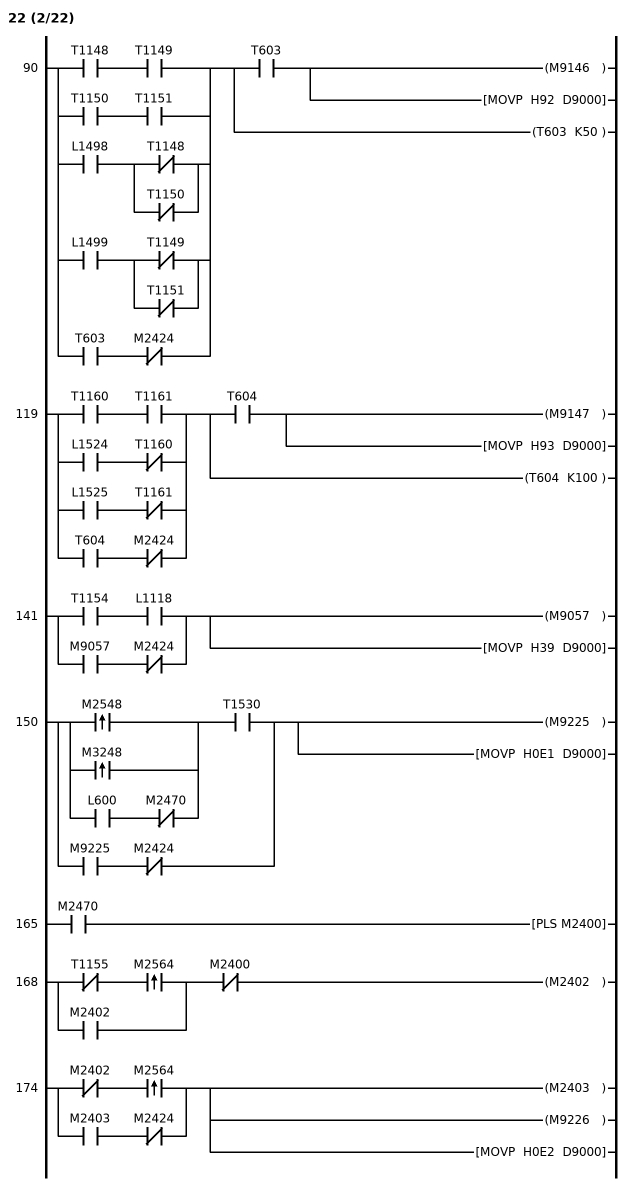
90    LD      T1148
      AND     T1149
      LD      T1150
      AND     T1151
      ORB
      LD      L1498
      LDI     T1148
      ORI     T1150
      ANB
      ORB
      LD      L1499
      LDI     T1149
      ORI     T1151
      ANB
      ORB
      LD      T603
      ANI     M2424
      ORB
      MPS
      AND     T603
      OUT     M9146
      MOVP    H92 D9000
      MPP
      OUT     T603 K50
119   LD      T1160
      AND     T1161
      LD      L1524
      ANI     T1160
      ORB
      LD      L1525
      ANI     T1161
      ORB
      LD      T604
      ANI     M2424
      ORB
      MPS
      AND     T604
      OUT     M9147
      MOVP    H93 D9000
      MPP
      OUT     T604 K100
141   LD      T1154
      AND     L1118
      LD      M9057
      ANI     M2424
      ORB
      OUT     M9057
      MOVP    H39 D9000
150   LDP     M2548
      ORP     M3248
      LD      L600
      ANI     M2470
      ORB
      AND     T1530
      LD      M9225
      ANI     M2424
      ORB
      OUT     M9225
      MOVP    H0E1 D9000
165   LD      M2470
      PLS     M2400
168   LDI     T1155
      ANDP    M2564
      OR      M2402
      ANI     M2400
      OUT     M2402
174   LDI     M2402
      ANDP    M2564
      LD      M2403
      ANI     M2424
      ORB
      OUT     M2403
      OUT     M9226
      MOVP    H0E2 D9000
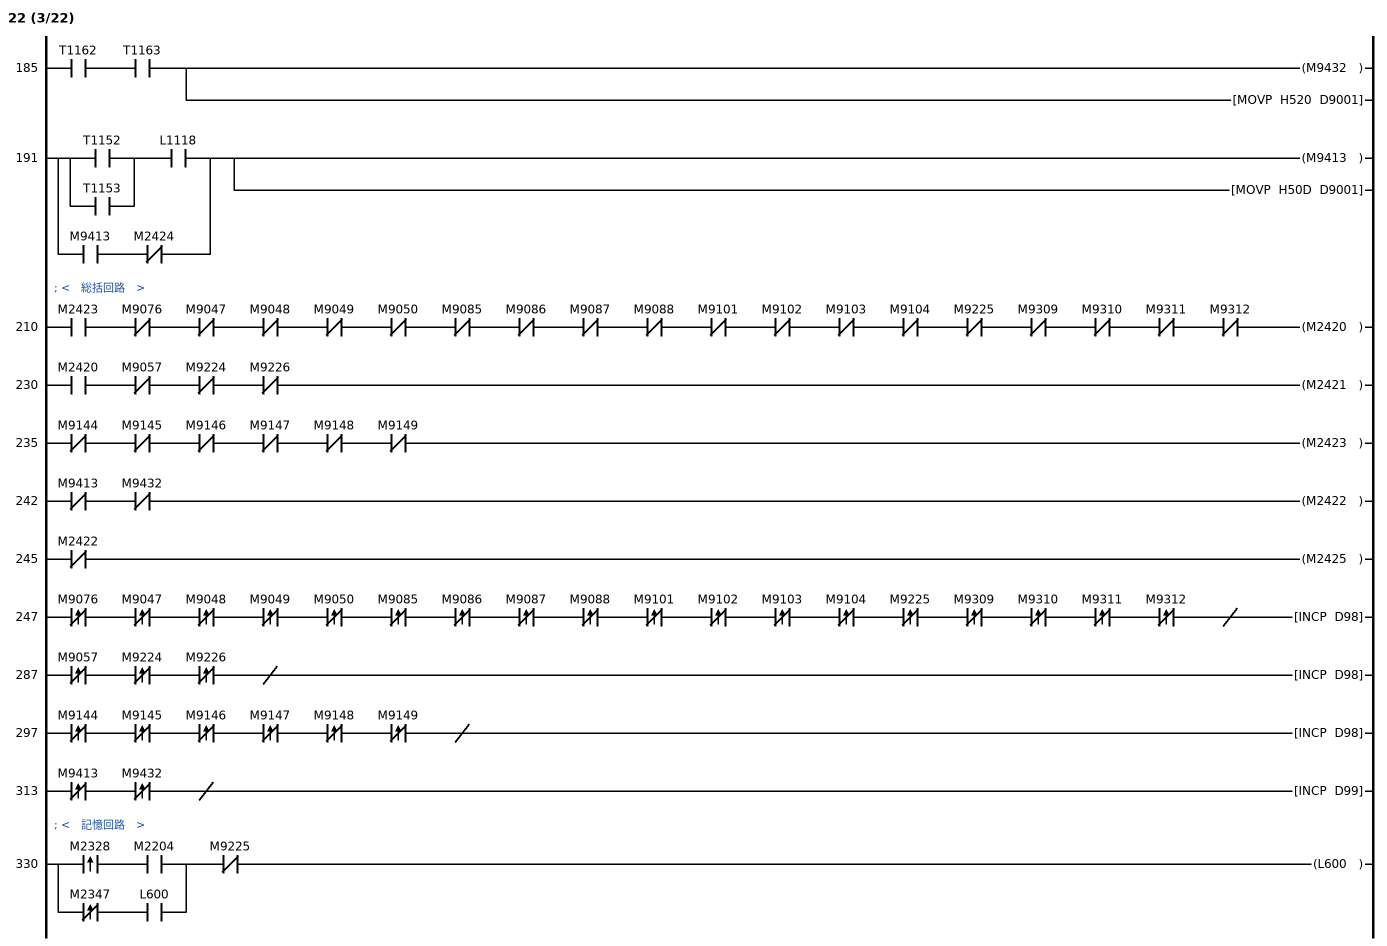
185   LD      T1162
      AND     T1163
      OUT     M9432
      MOVP    H520 D9001
191   LD      T1152
      OR      T1153
      AND     L1118
      LD      M9413
      ANI     M2424
      ORB
      OUT     M9413
      MOVP    H50D D9001
; <　総括回路　>
210   LD      M2423
      ANI     M9076
      ANI     M9047
      ANI     M9048
      ANI     M9049
      ANI     M9050
      ANI     M9085
      ANI     M9086
      ANI     M9087
      ANI     M9088
      ANI     M9101
      ANI     M9102
      ANI     M9103
      ANI     M9104
      ANI     M9225
      ANI     M9309
      ANI     M9310
      ANI     M9311
      ANI     M9312
      OUT     M2420
230   LD      M2420
      ANI     M9057
      ANI     M9224
      ANI     M9226
      OUT     M2421
235   LDI     M9144
      ANI     M9145
      ANI     M9146
      ANI     M9147
      ANI     M9148
      ANI     M9149
      OUT     M2423
242   LDI     M9413
      ANI     M9432
      OUT     M2422
245   LDI     M2422
      OUT     M2425
247   LDPI    M9076
      ANDPI   M9047
      ANDPI   M9048
      ANDPI   M9049
      ANDPI   M9050
      ANDPI   M9085
      ANDPI   M9086
      ANDPI   M9087
      ANDPI   M9088
      ANDPI   M9101
      ANDPI   M9102
      ANDPI   M9103
      ANDPI   M9104
      ANDPI   M9225
      ANDPI   M9309
      ANDPI   M9310
      ANDPI   M9311
      ANDPI   M9312
      INV
      INCP    D98
287   LDPI    M9057
      ANDPI   M9224
      ANDPI   M9226
      INV
      INCP    D98
297   LDPI    M9144
      ANDPI   M9145
      ANDPI   M9146
      ANDPI   M9147
      ANDPI   M9148
      ANDPI   M9149
      INV
      INCP    D98
313   LDPI    M9413
      ANDPI   M9432
      INV
      INCP    D99
; <　記憶回路　>
330   LDP     M2328
      AND     M2204
      LDPI    M2347
      AND     L600
      ORB
      ANI     M9225
      OUT     L600
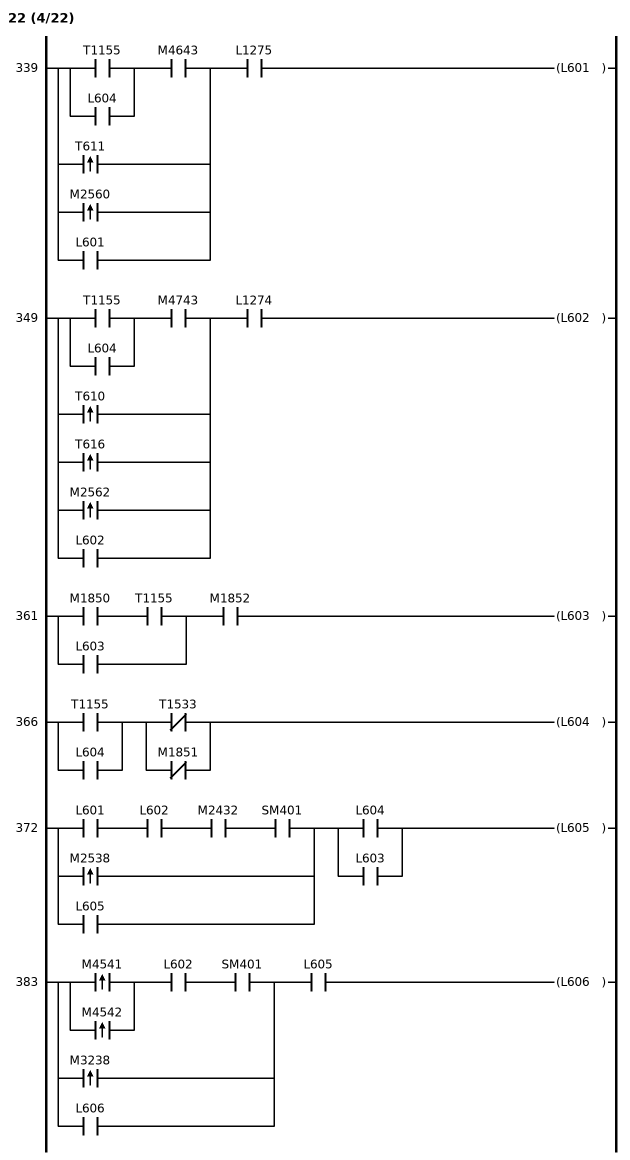
339   LD      T1155
      OR      L604
      AND     M4643
      ORP     T611
      ORP     M2560
      OR      L601
      AND     L1275
      OUT     L601
349   LD      T1155
      OR      L604
      AND     M4743
      ORP     T610
      ORP     T616
      ORP     M2562
      OR      L602
      AND     L1274
      OUT     L602
361   LD      M1850
      AND     T1155
      OR      L603
      AND     M1852
      OUT     L603
366   LD      T1155
      OR      L604
      LDI     T1533
      ORI     M1851
      ANB
      OUT     L604
372   LD      L601
      AND     L602
      AND     M2432
      AND     SM401
      ORP     M2538
      OR      L605
      LD      L604
      OR      L603
      ANB
      OUT     L605
383   LDP     M4541
      ORP     M4542
      AND     L602
      AND     SM401
      ORP     M3238
      OR      L606
      AND     L605
      OUT     L606
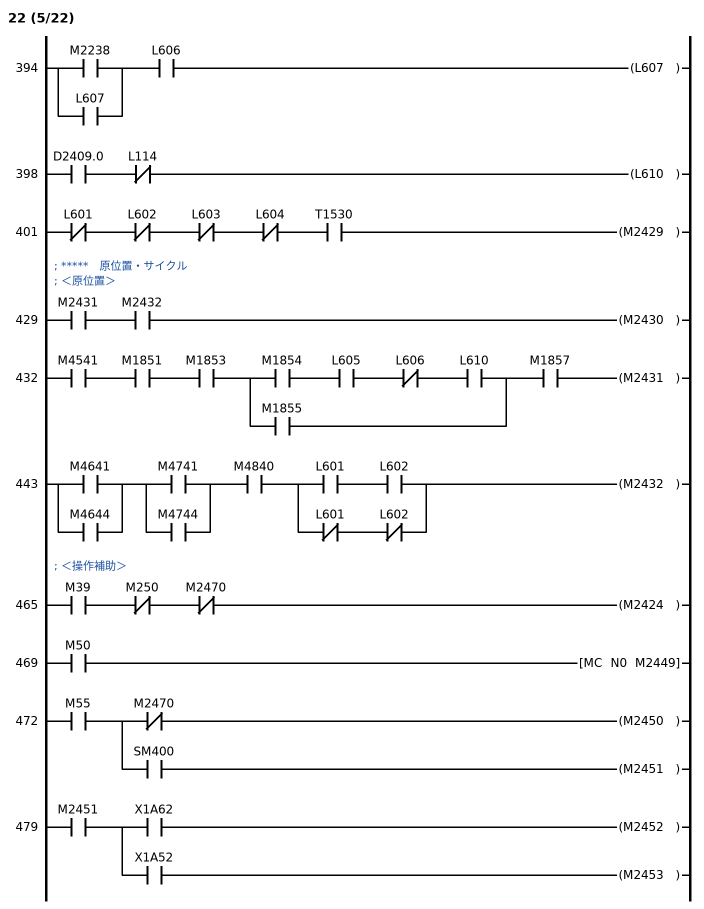
394   LD      M2238
      OR      L607
      AND     L606
      OUT     L607
398   LD      D2409.0
      ANI     L114
      OUT     L610
401   LDI     L601
      ANI     L602
      ANI     L603
      ANI     L604
      AND     T1530
      OUT     M2429
; *****　原位置・サイクル
; ＜原位置＞
429   LD      M2431
      AND     M2432
      OUT     M2430
432   LD      M4541
      AND     M1851
      AND     M1853
      LD      M1854
      AND     L605
      ANI     L606
      AND     L610
      OR      M1855
      ANB
      AND     M1857
      OUT     M2431
443   LD      M4641
      OR      M4644
      LD      M4741
      OR      M4744
      ANB
      AND     M4840
      LD      L601
      AND     L602
      LDI     L601
      ANI     L602
      ORB
      ANB
      OUT     M2432
; ＜操作補助＞
465   LD      M39
      ANI     M250
      ANI     M2470
      OUT     M2424
469   LD      M50
      MC      N0 M2449
472   LD      M55
      MPS
      ANI     M2470
      OUT     M2450
      MPP
      AND     SM400
      OUT     M2451
479   LD      M2451
      MPS
      AND     X1A62
      OUT     M2452
      MPP
      AND     X1A52
      OUT     M2453
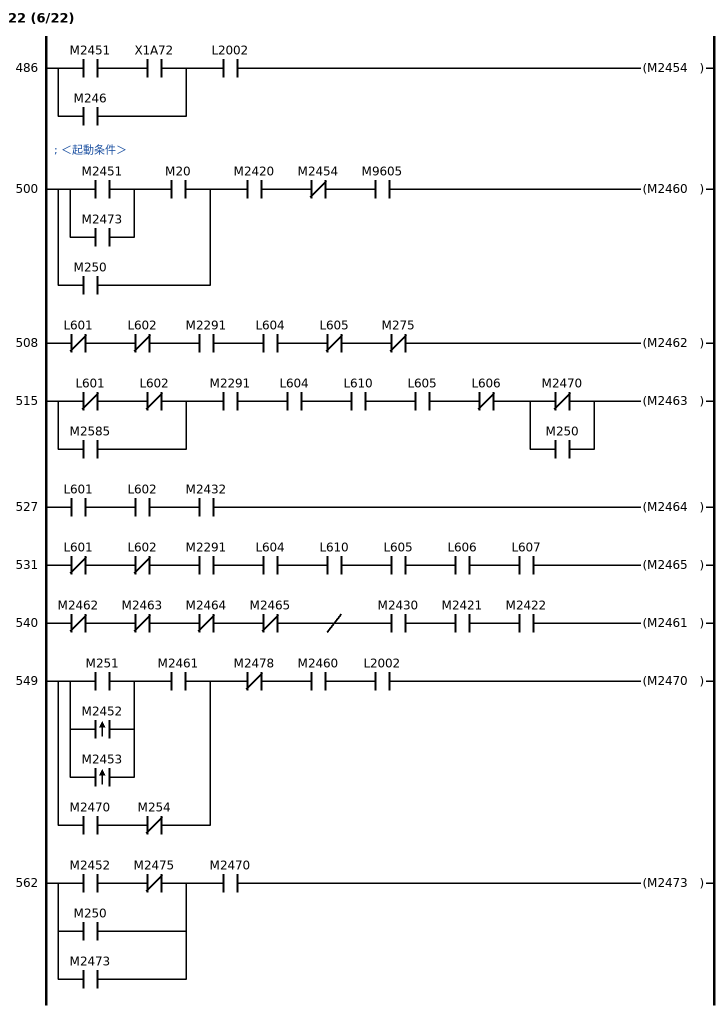
486   LD      M2451
      AND     X1A72
      OR      M246
      AND     L2002
      OUT     M2454
; ＜起動条件＞
500   LD      M2451
      OR      M2473
      AND     M20
      OR      M250
      AND     M2420
      ANI     M2454
      AND     M9605
      OUT     M2460
508   LDI     L601
      ANI     L602
      AND     M2291
      AND     L604
      ANI     L605
      ANI     M275
      OUT     M2462
515   LDI     L601
      ANI     L602
      OR      M2585
      AND     M2291
      AND     L604
      AND     L610
      AND     L605
      ANI     L606
      LDI     M2470
      OR      M250
      ANB
      OUT     M2463
527   LD      L601
      AND     L602
      AND     M2432
      OUT     M2464
531   LDI     L601
      ANI     L602
      AND     M2291
      AND     L604
      AND     L610
      AND     L605
      AND     L606
      AND     L607
      OUT     M2465
540   LDI     M2462
      ANI     M2463
      ANI     M2464
      ANI     M2465
      INV
      AND     M2430
      AND     M2421
      AND     M2422
      OUT     M2461
549   LD      M251
      ORP     M2452
      ORP     M2453
      AND     M2461
      LD      M2470
      ANI     M254
      ORB
      ANI     M2478
      AND     M2460
      AND     L2002
      OUT     M2470
562   LD      M2452
      ANI     M2475
      OR      M250
      OR      M2473
      AND     M2470
      OUT     M2473
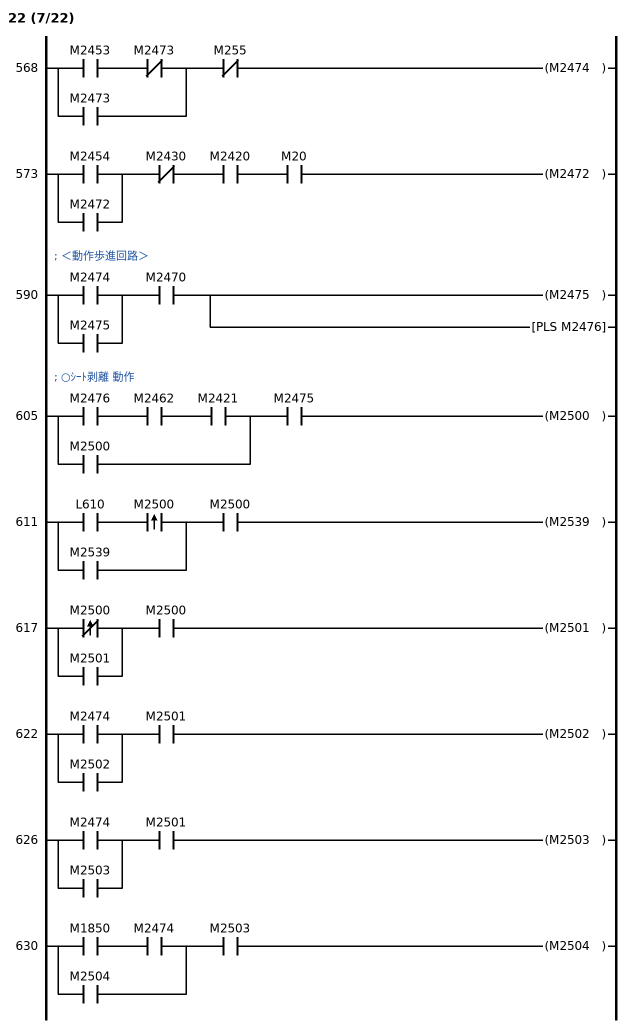
568   LD      M2453
      ANI     M2473
      OR      M2473
      ANI     M255
      OUT     M2474
573   LD      M2454
      OR      M2472
      ANI     M2430
      AND     M2420
      AND     M20
      OUT     M2472
; ＜動作歩進回路＞
590   LD      M2474
      OR      M2475
      AND     M2470
      OUT     M2475
      PLS     M2476
; ○ｼｰﾄ剥離 動作
605   LD      M2476
      AND     M2462
      AND     M2421
      OR      M2500
      AND     M2475
      OUT     M2500
611   LD      L610
      ANDP    M2500
      OR      M2539
      AND     M2500
      OUT     M2539
617   LDPI    M2500
      OR      M2501
      AND     M2500
      OUT     M2501
622   LD      M2474
      OR      M2502
      AND     M2501
      OUT     M2502
626   LD      M2474
      OR      M2503
      AND     M2501
      OUT     M2503
630   LD      M1850
      AND     M2474
      OR      M2504
      AND     M2503
      OUT     M2504
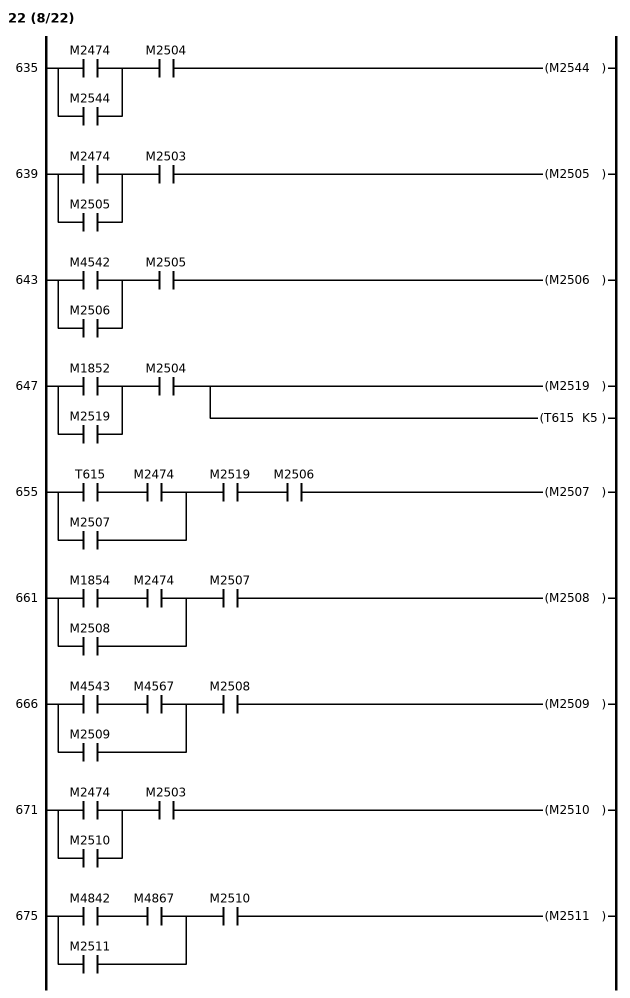
635   LD      M2474
      OR      M2544
      AND     M2504
      OUT     M2544
639   LD      M2474
      OR      M2505
      AND     M2503
      OUT     M2505
643   LD      M4542
      OR      M2506
      AND     M2505
      OUT     M2506
647   LD      M1852
      OR      M2519
      AND     M2504
      OUT     M2519
      OUT     T615 K5
655   LD      T615
      AND     M2474
      OR      M2507
      AND     M2519
      AND     M2506
      OUT     M2507
661   LD      M1854
      AND     M2474
      OR      M2508
      AND     M2507
      OUT     M2508
666   LD      M4543
      AND     M4567
      OR      M2509
      AND     M2508
      OUT     M2509
671   LD      M2474
      OR      M2510
      AND     M2503
      OUT     M2510
675   LD      M4842
      AND     M4867
      OR      M2511
      AND     M2510
      OUT     M2511
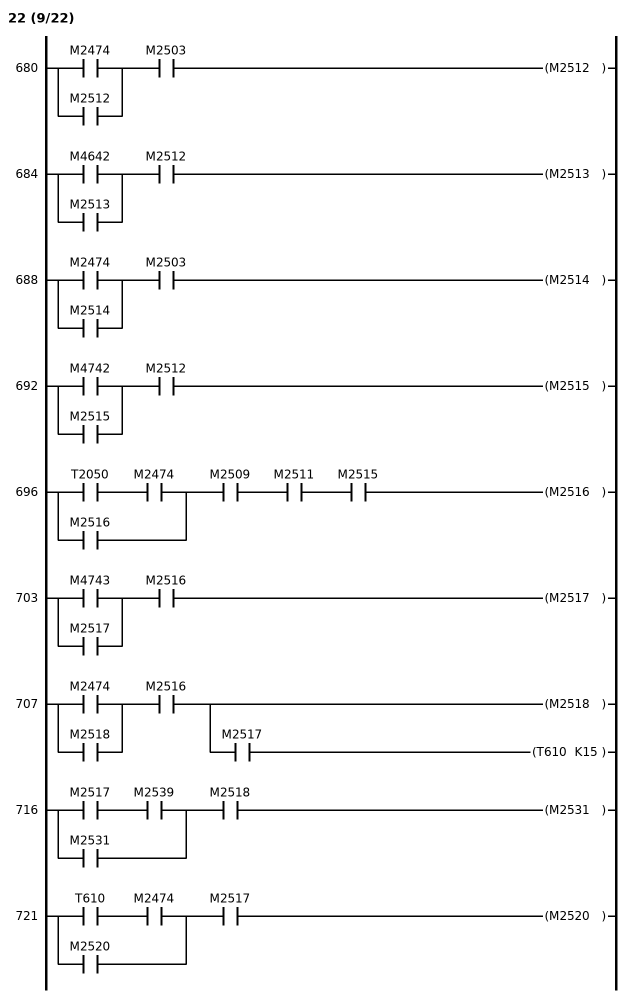
680   LD      M2474
      OR      M2512
      AND     M2503
      OUT     M2512
684   LD      M4642
      OR      M2513
      AND     M2512
      OUT     M2513
688   LD      M2474
      OR      M2514
      AND     M2503
      OUT     M2514
692   LD      M4742
      OR      M2515
      AND     M2512
      OUT     M2515
696   LD      T2050
      AND     M2474
      OR      M2516
      AND     M2509
      AND     M2511
      AND     M2515
      OUT     M2516
703   LD      M4743
      OR      M2517
      AND     M2516
      OUT     M2517
707   LD      M2474
      OR      M2518
      AND     M2516
      OUT     M2518
      AND     M2517
      OUT     T610 K15
716   LD      M2517
      AND     M2539
      OR      M2531
      AND     M2518
      OUT     M2531
721   LD      T610
      AND     M2474
      OR      M2520
      AND     M2517
      OUT     M2520
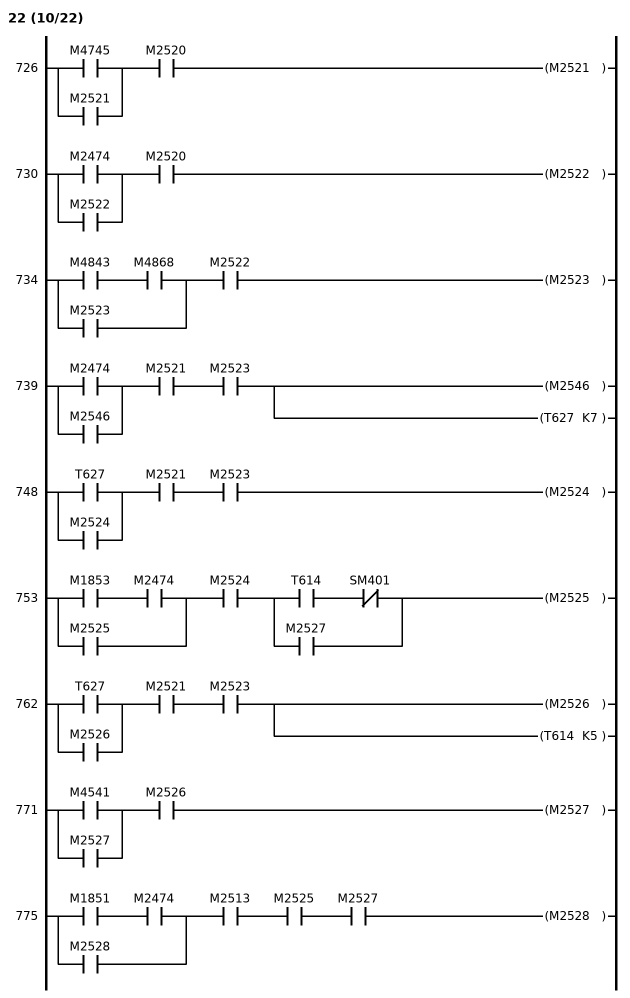
726   LD      M4745
      OR      M2521
      AND     M2520
      OUT     M2521
730   LD      M2474
      OR      M2522
      AND     M2520
      OUT     M2522
734   LD      M4843
      AND     M4868
      OR      M2523
      AND     M2522
      OUT     M2523
739   LD      M2474
      OR      M2546
      AND     M2521
      AND     M2523
      OUT     M2546
      OUT     T627 K7
748   LD      T627
      OR      M2524
      AND     M2521
      AND     M2523
      OUT     M2524
753   LD      M1853
      AND     M2474
      OR      M2525
      AND     M2524
      LD      T614
      ANI     SM401
      OR      M2527
      ANB
      OUT     M2525
762   LD      T627
      OR      M2526
      AND     M2521
      AND     M2523
      OUT     M2526
      OUT     T614 K5
771   LD      M4541
      OR      M2527
      AND     M2526
      OUT     M2527
775   LD      M1851
      AND     M2474
      OR      M2528
      AND     M2513
      AND     M2525
      AND     M2527
      OUT     M2528
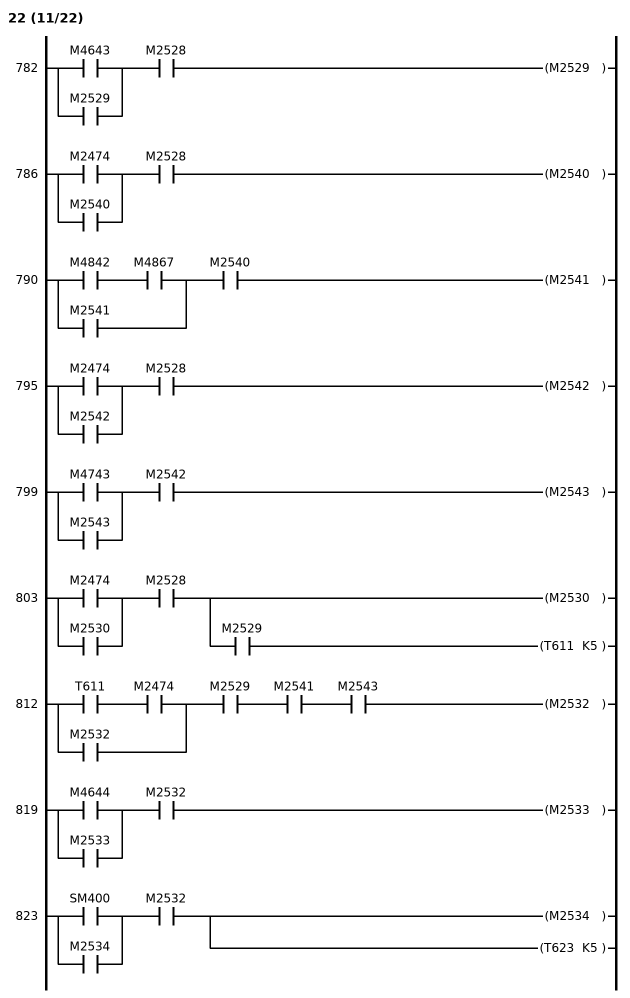
782   LD      M4643
      OR      M2529
      AND     M2528
      OUT     M2529
786   LD      M2474
      OR      M2540
      AND     M2528
      OUT     M2540
790   LD      M4842
      AND     M4867
      OR      M2541
      AND     M2540
      OUT     M2541
795   LD      M2474
      OR      M2542
      AND     M2528
      OUT     M2542
799   LD      M4743
      OR      M2543
      AND     M2542
      OUT     M2543
803   LD      M2474
      OR      M2530
      AND     M2528
      OUT     M2530
      AND     M2529
      OUT     T611 K5
812   LD      T611
      AND     M2474
      OR      M2532
      AND     M2529
      AND     M2541
      AND     M2543
      OUT     M2532
819   LD      M4644
      OR      M2533
      AND     M2532
      OUT     M2533
823   LD      SM400
      OR      M2534
      AND     M2532
      OUT     M2534
      OUT     T623 K5
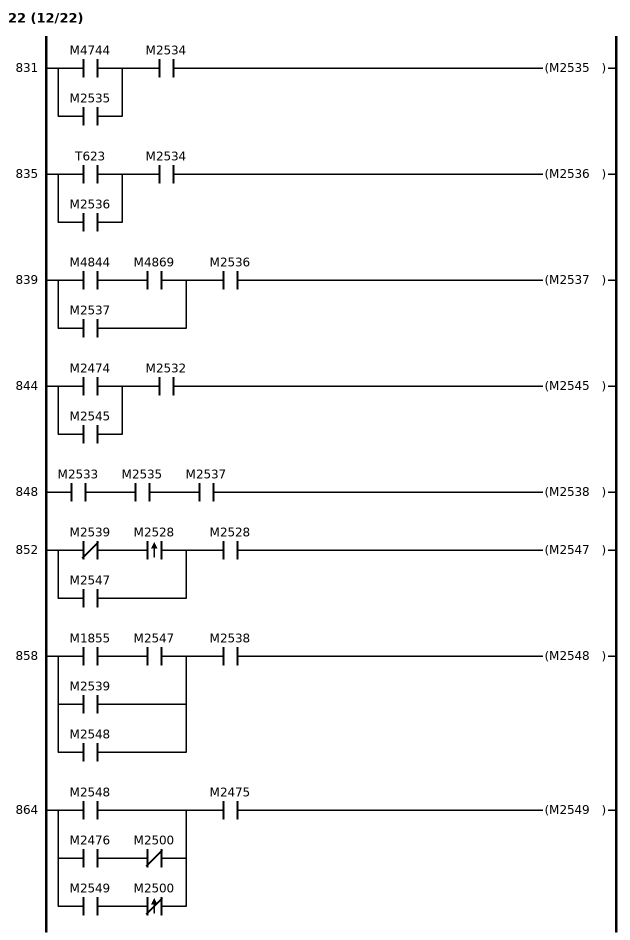
831   LD      M4744
      OR      M2535
      AND     M2534
      OUT     M2535
835   LD      T623
      OR      M2536
      AND     M2534
      OUT     M2536
839   LD      M4844
      AND     M4869
      OR      M2537
      AND     M2536
      OUT     M2537
844   LD      M2474
      OR      M2545
      AND     M2532
      OUT     M2545
848   LD      M2533
      AND     M2535
      AND     M2537
      OUT     M2538
852   LDI     M2539
      ANDP    M2528
      OR      M2547
      AND     M2528
      OUT     M2547
858   LD      M1855
      AND     M2547
      OR      M2539
      OR      M2548
      AND     M2538
      OUT     M2548
864   LD      M2548
      LD      M2476
      ANI     M2500
      ORB
      LD      M2549
      ANDPI   M2500
      ORB
      AND     M2475
      OUT     M2549
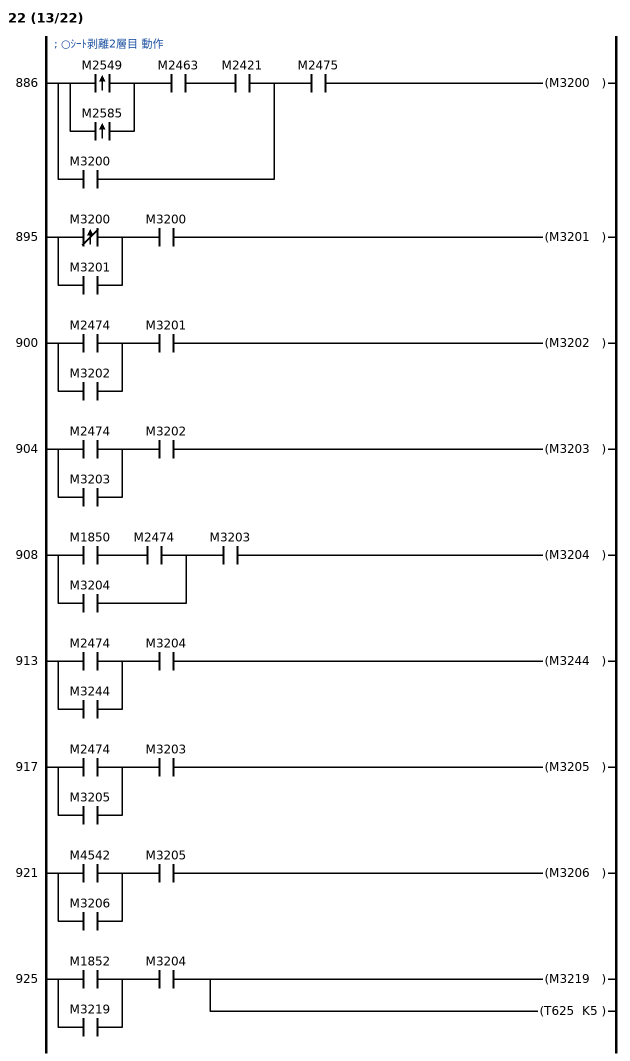
; ○ｼｰﾄ剥離2層目 動作
886   LDP     M2549
      ORP     M2585
      AND     M2463
      AND     M2421
      OR      M3200
      AND     M2475
      OUT     M3200
895   LDPI    M3200
      OR      M3201
      AND     M3200
      OUT     M3201
900   LD      M2474
      OR      M3202
      AND     M3201
      OUT     M3202
904   LD      M2474
      OR      M3203
      AND     M3202
      OUT     M3203
908   LD      M1850
      AND     M2474
      OR      M3204
      AND     M3203
      OUT     M3204
913   LD      M2474
      OR      M3244
      AND     M3204
      OUT     M3244
917   LD      M2474
      OR      M3205
      AND     M3203
      OUT     M3205
921   LD      M4542
      OR      M3206
      AND     M3205
      OUT     M3206
925   LD      M1852
      OR      M3219
      AND     M3204
      OUT     M3219
      OUT     T625 K5
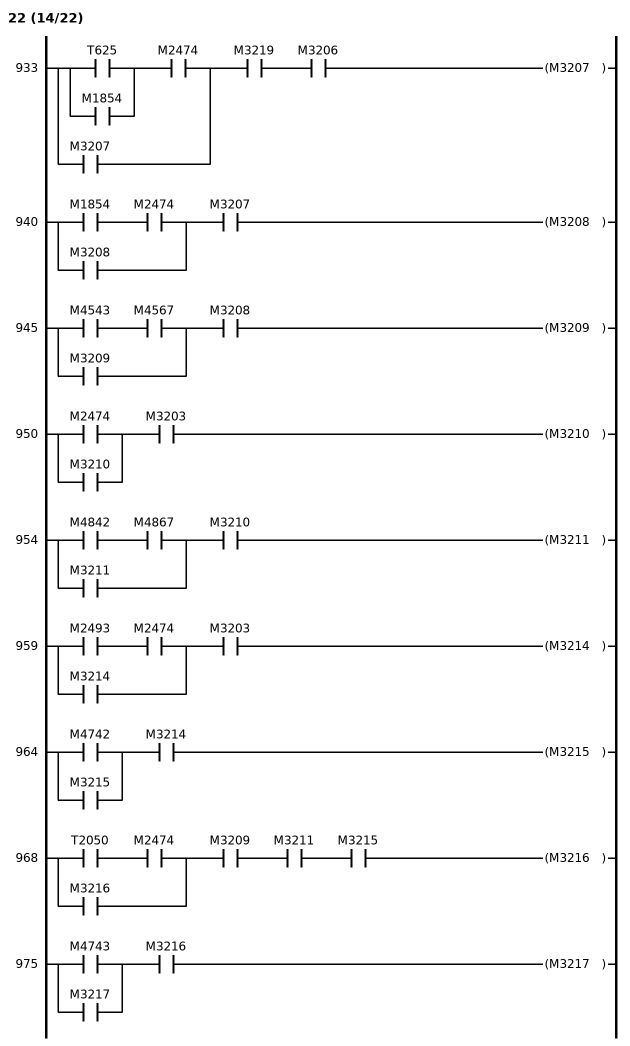
933   LD      T625
      OR      M1854
      AND     M2474
      OR      M3207
      AND     M3219
      AND     M3206
      OUT     M3207
940   LD      M1854
      AND     M2474
      OR      M3208
      AND     M3207
      OUT     M3208
945   LD      M4543
      AND     M4567
      OR      M3209
      AND     M3208
      OUT     M3209
950   LD      M2474
      OR      M3210
      AND     M3203
      OUT     M3210
954   LD      M4842
      AND     M4867
      OR      M3211
      AND     M3210
      OUT     M3211
959   LD      M2493
      AND     M2474
      OR      M3214
      AND     M3203
      OUT     M3214
964   LD      M4742
      OR      M3215
      AND     M3214
      OUT     M3215
968   LD      T2050
      AND     M2474
      OR      M3216
      AND     M3209
      AND     M3211
      AND     M3215
      OUT     M3216
975   LD      M4743
      OR      M3217
      AND     M3216
      OUT     M3217
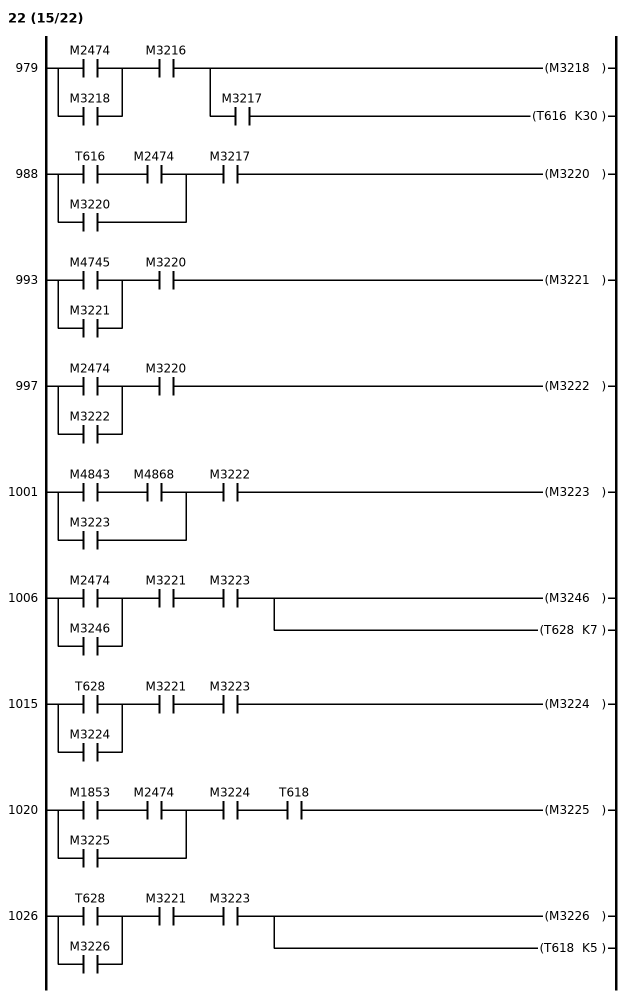
979   LD      M2474
      OR      M3218
      AND     M3216
      OUT     M3218
      AND     M3217
      OUT     T616 K30
988   LD      T616
      AND     M2474
      OR      M3220
      AND     M3217
      OUT     M3220
993   LD      M4745
      OR      M3221
      AND     M3220
      OUT     M3221
997   LD      M2474
      OR      M3222
      AND     M3220
      OUT     M3222
1001  LD      M4843
      AND     M4868
      OR      M3223
      AND     M3222
      OUT     M3223
1006  LD      M2474
      OR      M3246
      AND     M3221
      AND     M3223
      OUT     M3246
      OUT     T628 K7
1015  LD      T628
      OR      M3224
      AND     M3221
      AND     M3223
      OUT     M3224
1020  LD      M1853
      AND     M2474
      OR      M3225
      AND     M3224
      AND     T618
      OUT     M3225
1026  LD      T628
      OR      M3226
      AND     M3221
      AND     M3223
      OUT     M3226
      OUT     T618 K5
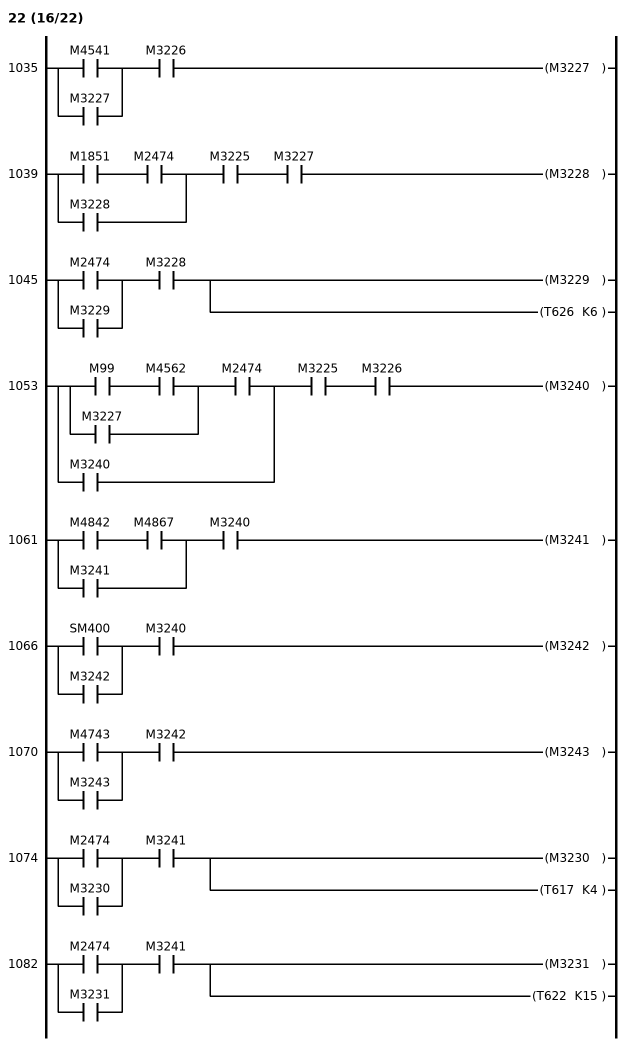
1035  LD      M4541
      OR      M3227
      AND     M3226
      OUT     M3227
1039  LD      M1851
      AND     M2474
      OR      M3228
      AND     M3225
      AND     M3227
      OUT     M3228
1045  LD      M2474
      OR      M3229
      AND     M3228
      OUT     M3229
      OUT     T626 K6
1053  LD      M99
      AND     M4562
      OR      M3227
      AND     M2474
      OR      M3240
      AND     M3225
      AND     M3226
      OUT     M3240
1061  LD      M4842
      AND     M4867
      OR      M3241
      AND     M3240
      OUT     M3241
1066  LD      SM400
      OR      M3242
      AND     M3240
      OUT     M3242
1070  LD      M4743
      OR      M3243
      AND     M3242
      OUT     M3243
1074  LD      M2474
      OR      M3230
      AND     M3241
      OUT     M3230
      OUT     T617 K4
1082  LD      M2474
      OR      M3231
      AND     M3241
      OUT     M3231
      OUT     T622 K15
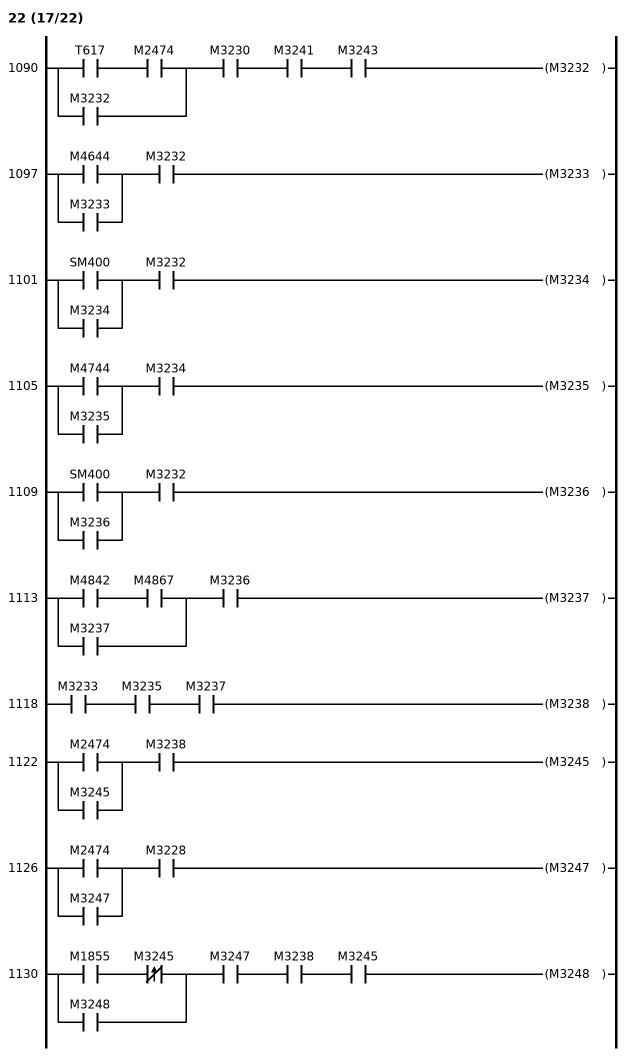
1090  LD      T617
      AND     M2474
      OR      M3232
      AND     M3230
      AND     M3241
      AND     M3243
      OUT     M3232
1097  LD      M4644
      OR      M3233
      AND     M3232
      OUT     M3233
1101  LD      SM400
      OR      M3234
      AND     M3232
      OUT     M3234
1105  LD      M4744
      OR      M3235
      AND     M3234
      OUT     M3235
1109  LD      SM400
      OR      M3236
      AND     M3232
      OUT     M3236
1113  LD      M4842
      AND     M4867
      OR      M3237
      AND     M3236
      OUT     M3237
1118  LD      M3233
      AND     M3235
      AND     M3237
      OUT     M3238
1122  LD      M2474
      OR      M3245
      AND     M3238
      OUT     M3245
1126  LD      M2474
      OR      M3247
      AND     M3228
      OUT     M3247
1130  LD      M1855
      ANDPI   M3245
      OR      M3248
      AND     M3247
      AND     M3238
      AND     M3245
      OUT     M3248
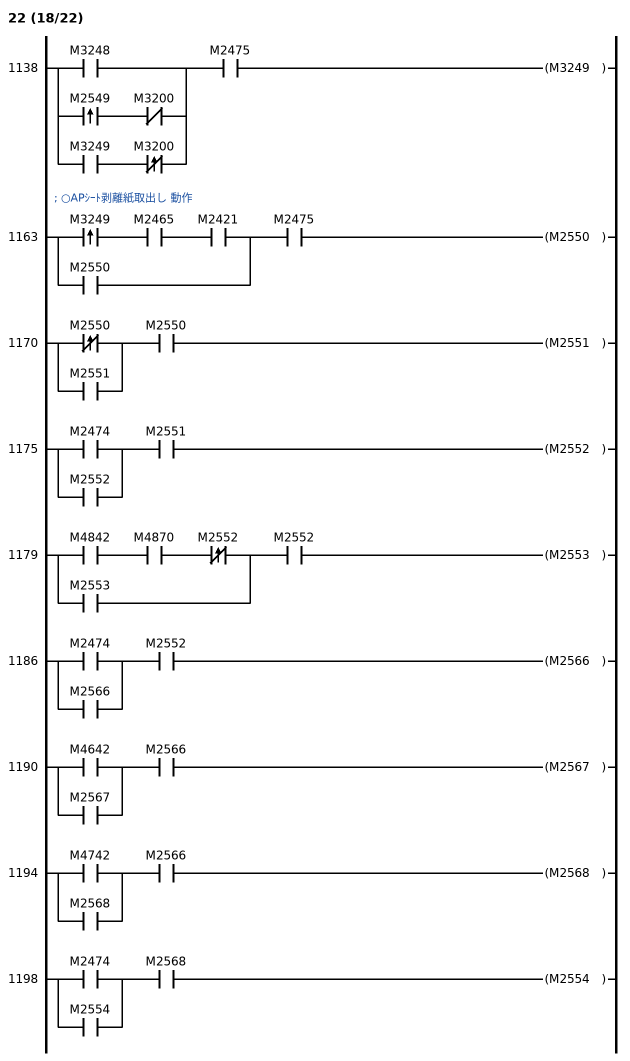
1138  LD      M3248
      LDP     M2549
      ANI     M3200
      ORB
      LD      M3249
      ANDPI   M3200
      ORB
      AND     M2475
      OUT     M3249
; ○APｼｰﾄ剥離紙取出し 動作
1163  LDP     M3249
      AND     M2465
      AND     M2421
      OR      M2550
      AND     M2475
      OUT     M2550
1170  LDPI    M2550
      OR      M2551
      AND     M2550
      OUT     M2551
1175  LD      M2474
      OR      M2552
      AND     M2551
      OUT     M2552
1179  LD      M4842
      AND     M4870
      ANDPI   M2552
      OR      M2553
      AND     M2552
      OUT     M2553
1186  LD      M2474
      OR      M2566
      AND     M2552
      OUT     M2566
1190  LD      M4642
      OR      M2567
      AND     M2566
      OUT     M2567
1194  LD      M4742
      OR      M2568
      AND     M2566
      OUT     M2568
1198  LD      M2474
      OR      M2554
      AND     M2568
      OUT     M2554
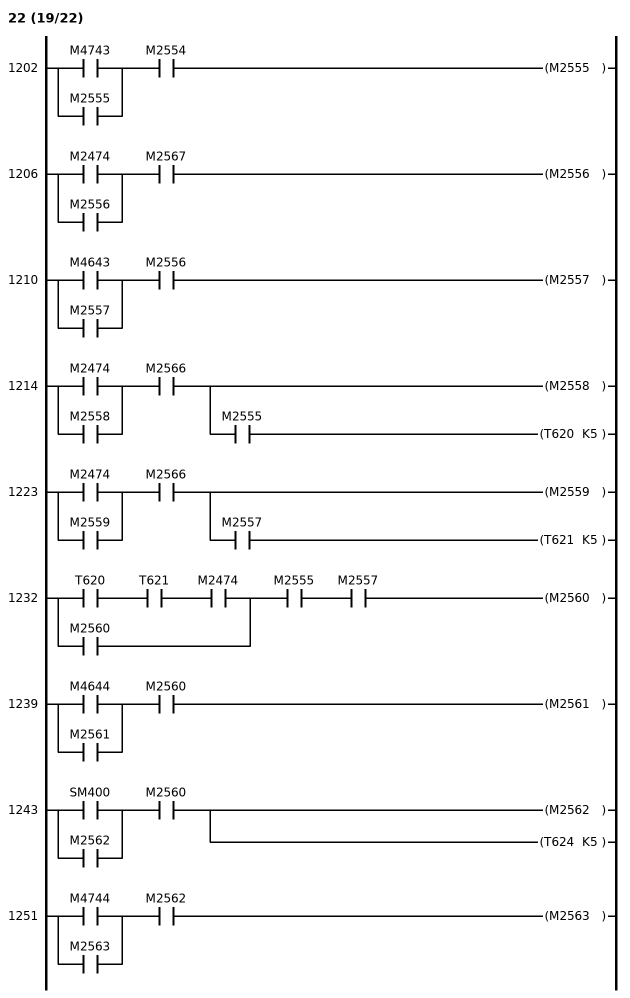
1202  LD      M4743
      OR      M2555
      AND     M2554
      OUT     M2555
1206  LD      M2474
      OR      M2556
      AND     M2567
      OUT     M2556
1210  LD      M4643
      OR      M2557
      AND     M2556
      OUT     M2557
1214  LD      M2474
      OR      M2558
      AND     M2566
      OUT     M2558
      AND     M2555
      OUT     T620 K5
1223  LD      M2474
      OR      M2559
      AND     M2566
      OUT     M2559
      AND     M2557
      OUT     T621 K5
1232  LD      T620
      AND     T621
      AND     M2474
      OR      M2560
      AND     M2555
      AND     M2557
      OUT     M2560
1239  LD      M4644
      OR      M2561
      AND     M2560
      OUT     M2561
1243  LD      SM400
      OR      M2562
      AND     M2560
      OUT     M2562
      OUT     T624 K5
1251  LD      M4744
      OR      M2563
      AND     M2562
      OUT     M2563
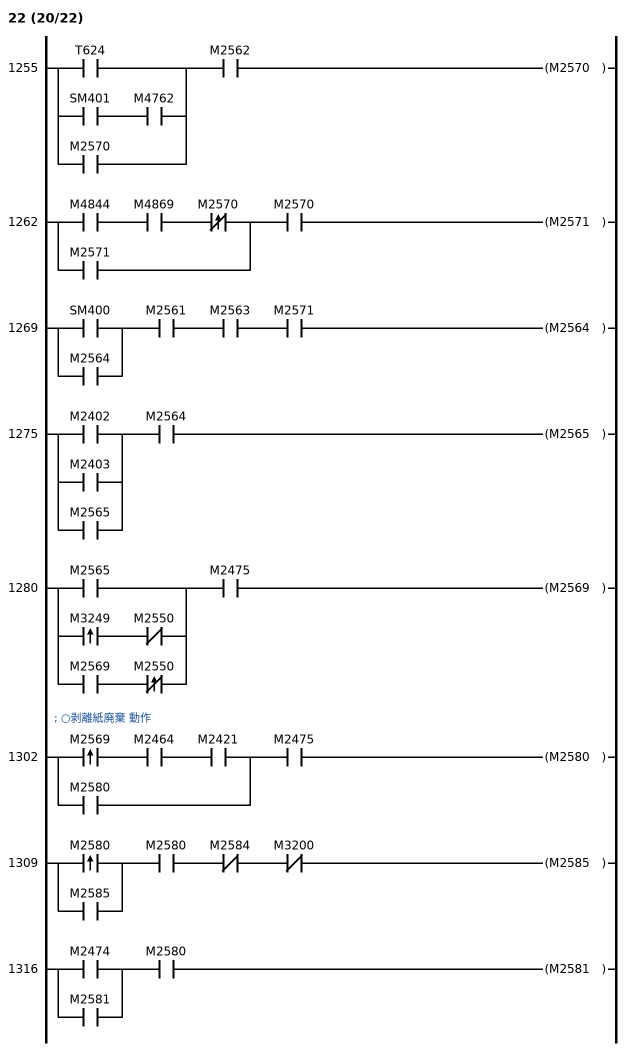
1255  LD      T624
      LD      SM401
      AND     M4762
      ORB
      OR      M2570
      AND     M2562
      OUT     M2570
1262  LD      M4844
      AND     M4869
      ANDPI   M2570
      OR      M2571
      AND     M2570
      OUT     M2571
1269  LD      SM400
      OR      M2564
      AND     M2561
      AND     M2563
      AND     M2571
      OUT     M2564
1275  LD      M2402
      OR      M2403
      OR      M2565
      AND     M2564
      OUT     M2565
1280  LD      M2565
      LDP     M3249
      ANI     M2550
      ORB
      LD      M2569
      ANDPI   M2550
      ORB
      AND     M2475
      OUT     M2569
; ○剥離紙廃棄 動作
1302  LDP     M2569
      AND     M2464
      AND     M2421
      OR      M2580
      AND     M2475
      OUT     M2580
1309  LDP     M2580
      OR      M2585
      AND     M2580
      ANI     M2584
      ANI     M3200
      OUT     M2585
1316  LD      M2474
      OR      M2581
      AND     M2580
      OUT     M2581
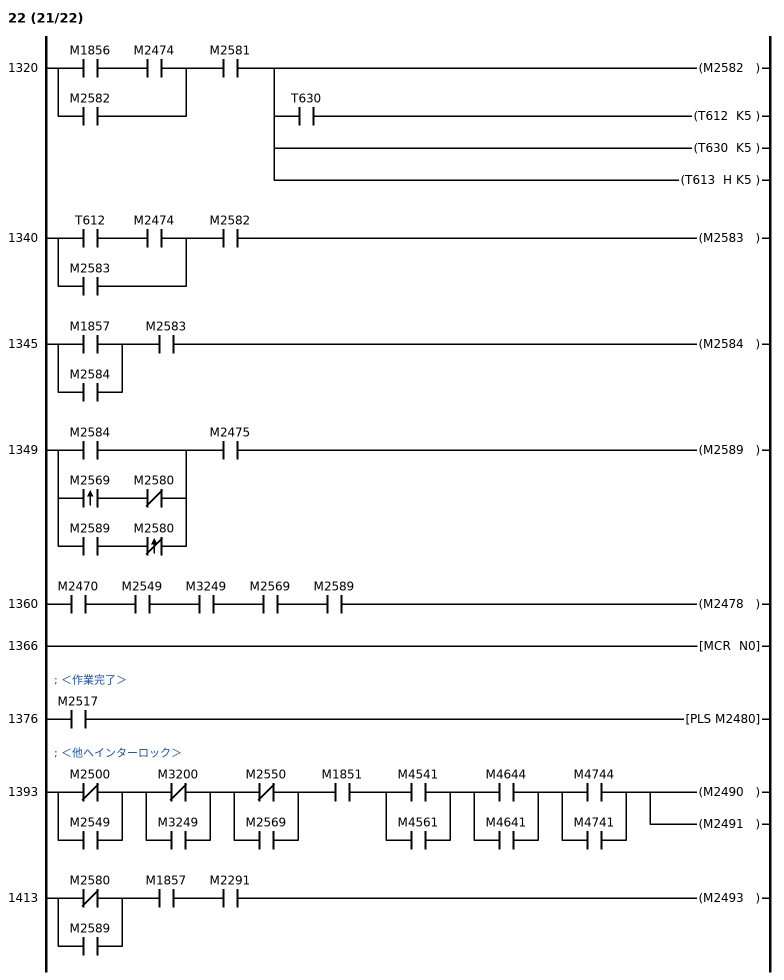
1320  LD      M1856
      AND     M2474
      OR      M2582
      AND     M2581
      OUT     M2582
      MPS
      AND     T630
      OUT     T612 K5
      MPP
      OUT     T630 K5
      OUTH    T613 K5
1340  LD      T612
      AND     M2474
      OR      M2583
      AND     M2582
      OUT     M2583
1345  LD      M1857
      OR      M2584
      AND     M2583
      OUT     M2584
1349  LD      M2584
      LDP     M2569
      ANI     M2580
      ORB
      LD      M2589
      ANDPI   M2580
      ORB
      AND     M2475
      OUT     M2589
1360  LD      M2470
      AND     M2549
      AND     M3249
      AND     M2569
      AND     M2589
      OUT     M2478
1366  MCR     N0
; ＜作業完了＞
1376  LD      M2517
      PLS     M2480
; ＜他へインターロック＞
1393  LDI     M2500
      OR      M2549
      LDI     M3200
      OR      M3249
      ANB
      LDI     M2550
      OR      M2569
      ANB
      AND     M1851
      LD      M4541
      OR      M4561
      ANB
      LD      M4644
      OR      M4641
      ANB
      LD      M4744
      OR      M4741
      ANB
      OUT     M2490
      OUT     M2491
1413  LDI     M2580
      OR      M2589
      AND     M1857
      AND     M2291
      OUT     M2493
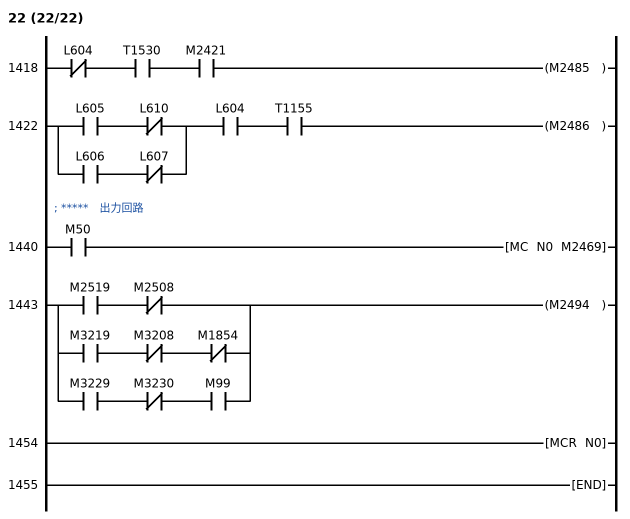
1418  LDI     L604
      AND     T1530
      AND     M2421
      OUT     M2485
1422  LD      L605
      ANI     L610
      LD      L606
      ANI     L607
      ORB
      AND     L604
      AND     T1155
      OUT     M2486
; *****　出力回路
1440  LD      M50
      MC      N0 M2469
1443  LD      M2519
      ANI     M2508
      LD      M3219
      ANI     M3208
      ANI     M1854
      ORB
      LD      M3229
      ANI     M3230
      AND     M99
      ORB
      OUT     M2494
1454  MCR     N0
1455  END
END_PROGRAM

PROGRAM 23
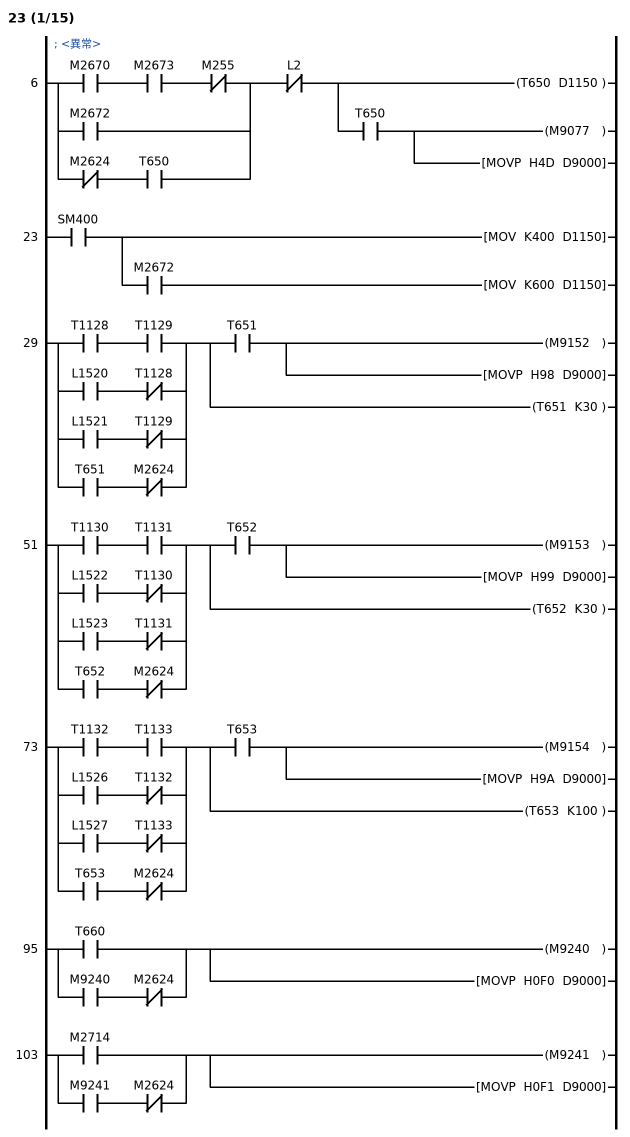
; <異常>
6     LD      M2670
      AND     M2673
      ANI     M255
      OR      M2672
      LDI     M2624
      AND     T650
      ORB
      ANI     L2
      OUT     T650 D1150
      AND     T650
      OUT     M9077
      MOVP    H4D D9000
23    LD      SM400
      MOV     K400 D1150
      AND     M2672
      MOV     K600 D1150
29    LD      T1128
      AND     T1129
      LD      L1520
      ANI     T1128
      ORB
      LD      L1521
      ANI     T1129
      ORB
      LD      T651
      ANI     M2624
      ORB
      MPS
      AND     T651
      OUT     M9152
      MOVP    H98 D9000
      MPP
      OUT     T651 K30
51    LD      T1130
      AND     T1131
      LD      L1522
      ANI     T1130
      ORB
      LD      L1523
      ANI     T1131
      ORB
      LD      T652
      ANI     M2624
      ORB
      MPS
      AND     T652
      OUT     M9153
      MOVP    H99 D9000
      MPP
      OUT     T652 K30
73    LD      T1132
      AND     T1133
      LD      L1526
      ANI     T1132
      ORB
      LD      L1527
      ANI     T1133
      ORB
      LD      T653
      ANI     M2624
      ORB
      MPS
      AND     T653
      OUT     M9154
      MOVP    H9A D9000
      MPP
      OUT     T653 K100
95    LD      T660
      LD      M9240
      ANI     M2624
      ORB
      OUT     M9240
      MOVP    H0F0 D9000
103   LD      M2714
      LD      M9241
      ANI     M2624
      ORB
      OUT     M9241
      MOVP    H0F1 D9000
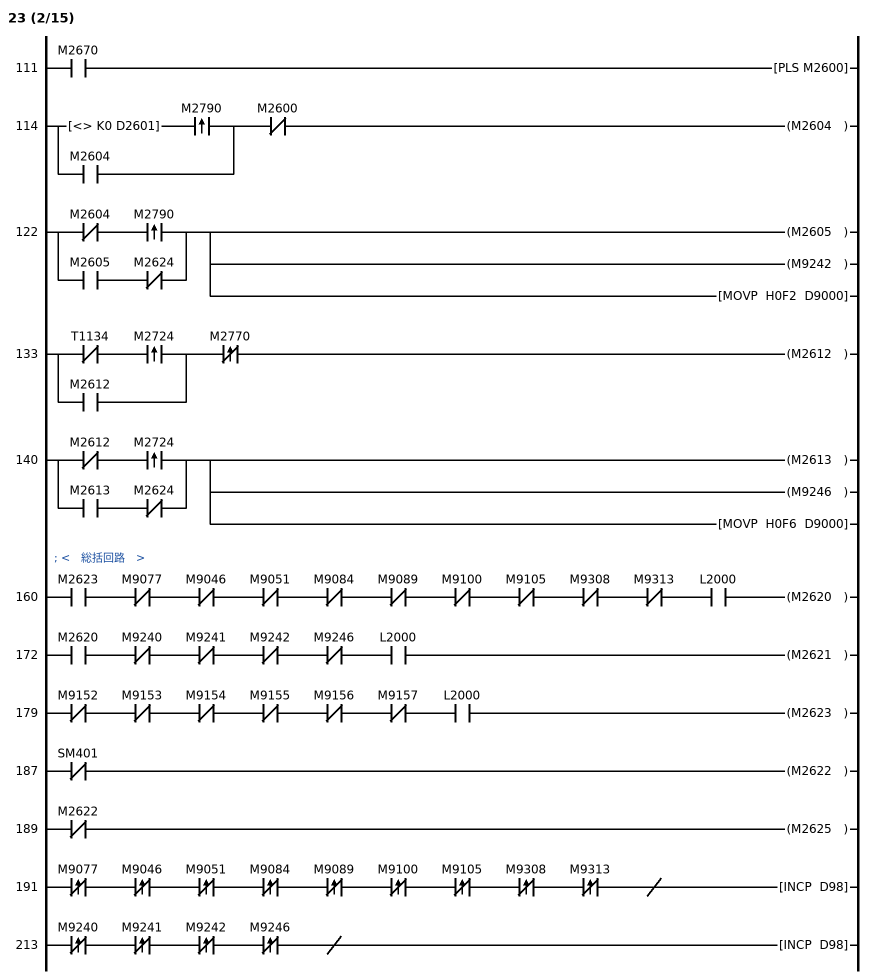
111   LD      M2670
      PLS     M2600
114   LD<>    K0 D2601
      ANDP    M2790
      OR      M2604
      ANI     M2600
      OUT     M2604
122   LDI     M2604
      ANDP    M2790
      LD      M2605
      ANI     M2624
      ORB
      OUT     M2605
      OUT     M9242
      MOVP    H0F2 D9000
133   LDI     T1134
      ANDP    M2724
      OR      M2612
      ANDPI   M2770
      OUT     M2612
140   LDI     M2612
      ANDP    M2724
      LD      M2613
      ANI     M2624
      ORB
      OUT     M2613
      OUT     M9246
      MOVP    H0F6 D9000
; <　総括回路　>
160   LD      M2623
      ANI     M9077
      ANI     M9046
      ANI     M9051
      ANI     M9084
      ANI     M9089
      ANI     M9100
      ANI     M9105
      ANI     M9308
      ANI     M9313
      AND     L2000
      OUT     M2620
172   LD      M2620
      ANI     M9240
      ANI     M9241
      ANI     M9242
      ANI     M9246
      AND     L2000
      OUT     M2621
179   LDI     M9152
      ANI     M9153
      ANI     M9154
      ANI     M9155
      ANI     M9156
      ANI     M9157
      AND     L2000
      OUT     M2623
187   LDI     SM401
      OUT     M2622
189   LDI     M2622
      OUT     M2625
191   LDPI    M9077
      ANDPI   M9046
      ANDPI   M9051
      ANDPI   M9084
      ANDPI   M9089
      ANDPI   M9100
      ANDPI   M9105
      ANDPI   M9308
      ANDPI   M9313
      INV
      INCP    D98
213   LDPI    M9240
      ANDPI   M9241
      ANDPI   M9242
      ANDPI   M9246
      INV
      INCP    D98
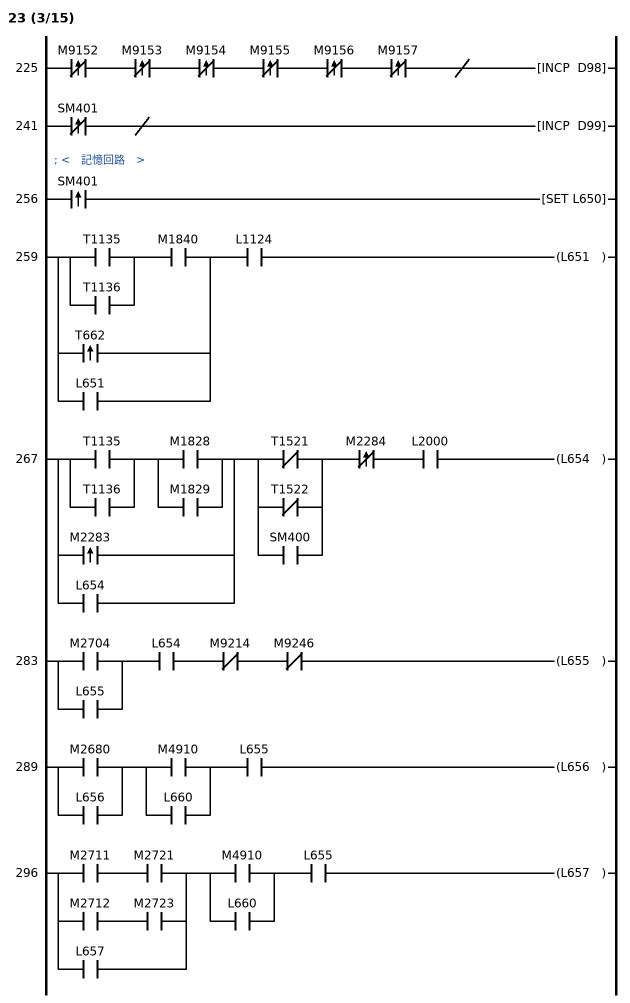
225   LDPI    M9152
      ANDPI   M9153
      ANDPI   M9154
      ANDPI   M9155
      ANDPI   M9156
      ANDPI   M9157
      INV
      INCP    D98
241   LDPI    SM401
      INV
      INCP    D99
; <　記憶回路　>
256   LDP     SM401
      SET     L650
259   LD      T1135
      OR      T1136
      AND     M1840
      ORP     T662
      OR      L651
      AND     L1124
      OUT     L651
267   LD      T1135
      OR      T1136
      LD      M1828
      OR      M1829
      ANB
      ORP     M2283
      OR      L654
      LDI     T1521
      ORI     T1522
      OR      SM400
      ANB
      ANDPI   M2284
      AND     L2000
      OUT     L654
283   LD      M2704
      OR      L655
      AND     L654
      ANI     M9214
      ANI     M9246
      OUT     L655
289   LD      M2680
      OR      L656
      LD      M4910
      OR      L660
      ANB
      AND     L655
      OUT     L656
296   LD      M2711
      AND     M2721
      LD      M2712
      AND     M2723
      ORB
      OR      L657
      LD      M4910
      OR      L660
      ANB
      AND     L655
      OUT     L657
